FUNCTION TryConvert_DWORD_TO_ULINT : BOOL
VAR_INPUT
	in : DWORD;
	out : REFERENCE TO ULINT;
END_VAR

out := DWORD_TO_ULINT(in);
TryConvert_DWORD_TO_ULINT := TRUE;

END_FUNCTION

(* stored: Version 1.1.0.1, ProductVersion 3.1.4024.12
   POU TryConvert_DWORD_TO_ULINT: Id {4179a511-159a-42c8-8762-c5de02ba67c2}, SpecialFunc None *)
